        ELSIF (PositionsMoverPresent[1] > 0) AND
              (PositionsMoverPresent[2] = 0)
        THEN
          nCycleMover               :=   PositionsMoverPresent[1];
          nAxisFirst[nCycleMover]   :=   2;
          nCycle                    := 120;
        END_IF

      120:  // X=360 Y=120 --> 2
        IF  (PositionsMoverPresent[3] = 0) AND
            (PositionsMoverPresent[2] > 0)
        THEN
          nCycleMover               :=   PositionsMoverPresent[2];
          nAxisFirst[nCycleMover]   :=   2;
          nCycle                    := 130;

        ELSIF (PositionsMoverPresent[1] = 0) AND
              (PositionsMoverPresent[3] > 0)
        THEN
          nCycleMover               :=   PositionsMoverPresent[3];
          nAxisFirst[nCycleMover]   :=   0;
          nCycle                    := 110;
        END_IF

      130:  // X=360, Y=600 --> 3
        IF  (PositionsMoverPresent[3] = 0) AND
            (PositionsMoverPresent[2] > 0)
        THEN
          nCycleMover               :=   PositionsMoverPresent[2];
          nAxisFirst[nCycleMover]   :=   2;
          nCycle                    := 110;

        ELSIF (PositionsMoverPresent[3] > 0) AND
              (PositionsMoverPresent[1] > 0)
        THEN
          nCycleMover               :=   PositionsMoverPresent[1];
          nAxisFirst[nCycleMover]   :=   2;
          nCycle                    := 120;
        END_IF
    END_CASE
END_CASE
//-------------------------------------------------------------------------------------------------
// reset movers
//-------------------------------------------------------------------------------------------------
CASE nCycle
OF
  900:
    _bCyclePause                          :=
    _bCycleStop                           :=
    _bCycleStart                          := FALSE;

    MoverCtrl[1].Cmd                      := E_MOVER_CTRL.MOVER_RESET;

    IF (MoverState[1].State = E_MOVER_STATE.MOVER_RESET + E_PROGRESS.PROGRESS_DONE)
    THEN
      nCycle                              := 910;
      MoverCtrl[1].Cmd          := E_MOVER_CTRL.MOVER_NULL;

    ELSIF (MoverState[1].State = E_MOVER_STATE.MOVER_RESET + E_PROGRESS.PROGRESS_ERROR)
    THEN
      MoverCtrl[1].Cmd          := E_MOVER_CTRL.MOVER_NULL;
    END_IF

  910:
    MoverCtrl[2].Cmd                      := E_MOVER_CTRL.MOVER_RESET;

    IF (MoverState[2].State = E_MOVER_STATE.MOVER_RESET + E_PROGRESS.PROGRESS_DONE)
    THEN
      nCycle                              := 920;
      MoverCtrl[2].Cmd          := E_MOVER_CTRL.MOVER_NULL;

    ELSIF (MoverState[2].State = E_MOVER_STATE.MOVER_RESET + E_PROGRESS.PROGRESS_ERROR)
    THEN
      MoverCtrl[2].Cmd          := E_MOVER_CTRL.MOVER_NULL;
    END_IF

  920:
    MoverCtrl[1].Cmd                      := E_MOVER_CTRL.MOVER_DISABLE;

    IF (MoverState[1].State = E_MOVER_STATE.MOVER_DISABLE + E_PROGRESS.PROGRESS_DONE)
    THEN
      nCycle                              := 930;
      MoverCtrl[1].Cmd          := E_MOVER_CTRL.MOVER_NULL;
    END_IF

  930:
    MoverCtrl[2].Cmd                      := E_MOVER_CTRL.MOVER_DISABLE;

    IF (MoverState[2].State = E_MOVER_STATE.MOVER_DISABLE + E_PROGRESS.PROGRESS_DONE)
    THEN
      IF (_wCycleReset = 0)
      THEN
        nCycle                            := 0;
      ELSE
        nCycle                            := 1000;
      END_IF
      MoverCtrl[2].Cmd          := E_MOVER_CTRL.MOVER_NULL;
    END_IF
END_CASE
//-------------------------------------------------------------------------------------------------
// recovery procedure
//-------------------------------------------------------------------------------------------------
CASE nCycle
OF
  1000:
    _wCycleReset                          := 0;
    // position check
    // mover must be in position at any station
    IF  (PositionsMoverPresent[1] > 0) AND
        (PositionsMoverPresent[2] > 0)
    THEN
      nCycleMover                         := PositionsMoverPresent[2];
      MoveData[nCycleMover]               := Positions[3];
      nAxisFirst[nCycleMover]             := 2;

      MoverCtrl[1].Cmd                    := E_MOVER_CTRL.MOVER_ENABLE;
      MoverCtrl[2].Cmd                    := E_MOVER_CTRL.MOVER_ENABLE;
  
      IF (MoverState[1].State = E_MOVER_STATE.MOVER_ENABLE + E_PROGRESS.PROGRESS_DONE) AND
         (MoverState[2].State = E_MOVER_STATE.MOVER_ENABLE + E_PROGRESS.PROGRESS_DONE)
      THEN
        nCycle                        := 1010;
      ELSE
        IF (MoverInfo[1].bMoverError) OR
           (MoverInfo[2].bMoverError)
        THEN
          nCycle                      := 900;
        END_IF
      END_IF

    ELSIF (PositionsMoverPresent[1] > 0) AND
          (PositionsMoverPresent[3] > 0)
    THEN
      nCycleMover                         := PositionsMoverPresent[1];
      MoveData[nCycleMover]               := Positions[2];
      nAxisFirst[nCycleMover]             := 2;

      MoverCtrl[1].Cmd                := E_MOVER_CTRL.MOVER_ENABLE;
      MoverCtrl[2].Cmd                := E_MOVER_CTRL.MOVER_ENABLE;
  
      IF (MoverState[1].State = E_MOVER_STATE.MOVER_ENABLE + E_PROGRESS.PROGRESS_DONE) AND
         (MoverState[2].State = E_MOVER_STATE.MOVER_ENABLE + E_PROGRESS.PROGRESS_DONE)
      THEN
        nCycle                        := 1010;
      ELSE
        IF (MoverInfo[1].bMoverError) OR
           (MoverInfo[2].bMoverError)
        THEN
          nCycle                      := 900;
        END_IF
      END_IF


    ELSIF (PositionsMoverPresent[2] > 0) AND
          (PositionsMoverPresent[3] > 0)
    THEN
      nCycleMover                         := PositionsMoverPresent[3];
      MoveData[nCycleMover]               := Positions[1];
      nAxisFirst[nCycleMover]             := 2;

      MoverCtrl[1].Cmd                := E_MOVER_CTRL.MOVER_ENABLE;
      MoverCtrl[2].Cmd                := E_MOVER_CTRL.MOVER_ENABLE;
  
      IF (MoverState[1].State = E_MOVER_STATE.MOVER_ENABLE + E_PROGRESS.PROGRESS_DONE) AND
         (MoverState[2].State = E_MOVER_STATE.MOVER_ENABLE + E_PROGRESS.PROGRESS_DONE)
      THEN
        nCycle                        := 1010;
      ELSE
        IF (MoverInfo[1].bMoverError) OR
           (MoverInfo[2].bMoverError)
        THEN
          nCycle                      := 900;
        END_IF
      END_IF
    END_IF

  1010:
      MoverCtrl[nCycleMover].Cmd    := E_MOVER_CTRL.MOVER_MOVE_TO_POS;
      IF (MoverState[nCycleMover].State = E_MOVER_STATE.MOVER_MOVE_TO_POS + E_PROGRESS.PROGRESS_ERROR)
      THEN
        nCycle                      := 900; // defaut error reaction: reset and switch off all movers

      ELSE
        IF (MoverState[nCycleMover].State = E_MOVER_STATE.MOVER_MOVE_TO_POS + E_PROGRESS.PROGRESS_DONE)
        THEN
          nCycle                    := 0;
        END_IF
      END_IF
END_CASE 
//-------------------------------------------------------------------------------------------------
//-------------------------------------------------------------------------------------------------
//-------------------------------------------------------------------------------------------------
//-------------------------------------------------------------------------------------------------
IF (_bClearAllAlarms)
THEN
  _bClearAllAlarms                  := FALSE;
  _hrEventLog                       := fbEventLogger.ClearAllAlarms(0, TRUE);
END_IF
//-------------------------------------------------------------------------------------------------
//-------------------------------------------------------------------------------------------------
IF (_bClearLoggedEvents)
THEN
  _bClearLoggedEvents               := fbEventLogger.ClearLoggedEvents(0);
END_IF
//-------------------------------------------------------------------------------------------------
//-------------------------------------------------------------------------------------------------
//-------------------------------------------------------------------------------------------------
//-------------------------------------------------------------------------------------------------

METHOD MoverInPositionXY : BOOL   // checks if XY position matches mover position
VAR_INPUT
  nMover              : DINT;
  stPosition          : ST_POS_XYC;
  rDelta              : ARRAY[1..2] OF LREAL;      // target window for X and Y
END_VAR
VAR
  bInPosition_X,
  bInPosition_Y       : BOOL;
END_VAR
VAR
//  rModPosC            : ARRAY[1..MAX_XPLANAR_MOVERS] OF LREAL;
END_VAR

IF NOT (nMover > 0) OR
   NOT (nMover < MAX_XPLANAR_MOVERS+1)
THEN
  RETURN;
END_IF


bInPosition_X         :=    (MoverInfo[nMover].rActPosX > stPosition.x - rDelta[1]) 
                        AND (MoverInfo[nMover].rActPosX < stPosition.x + rDelta[1]);

bInPosition_Y         :=    (MoverInfo[nMover].rActPosY > stPosition.y - rDelta[2]) 
                        AND (MoverInfo[nMover].rActPosY < stPosition.y + rDelta[2]);

rModPosC[nMover]      := Tc2_Math.LMOD(MoverInfo[nMover].rActPosC, 90.0);

IF (bInPosition_X AND bInPosition_Y)
THEN
  IF ((rModPosC[nMover]) <   5) AND
     ((rModPosC[nMover]) >  -5)
  THEN
    MoverInPositionXY := TRUE;
  ELSIF (ABS(rModPosC[nMover]) < 95) AND
        (ABS(rModPosC[nMover]) > 85)
  THEN
    MoverInPositionXY := TRUE;
  END_IF
END_IF
END_METHOD

END_PROGRAM

// ---- Mover/fb_MoverCtrl.TcPOU
//---------------------------------------------------------------------------------------------------------------
//
//  HAUD 2023.12.18
//
//  - XTS_TRAINING
//  - example project for setting up transport layer
//
//
//  fb_MoverCtrl
//  - accepts orders (E_MOVER_CTRL) via cyclic struct interface to execute
//  - interface struct  to extern control
//
//
//---------------------------------------------------------------------------------------------------------------
// This SOFTWARE is provided as an Exemple by THE PROVIDER "as is" and "with all faults." THE PROVIDER makes no 
// representations or warranties of any kind concerning the safety, suitability, lack of viruses, inaccuracies, 
// typographical errors, or other harmful components of this SOFTWARE. There are inherent dangers in the use of 
// any software, and you are solely responsible for determining whether this SOFTWARE is compatible with your 
// equipment and other software installed on your equipment. You are also solely responsible for the protection 
// of your equipment and backup of your data, and THE PROVIDER will not be liable for any damages you may suffer 
// in connection with using, modifying, or distributing this SOFTWARE.
//---------------------------------------------------------------------------------------------------------------
FUNCTION_BLOCK fb_MoverCtrl EXTENDS fb_Mover
VAR
  // Ctrl and State for executing commands
  _stCtrl           : REFERENCE TO ARRAY[1..MAX_XPLANAR_MOVERS] OF ST_MOVER_CTRL;
  _stState          : REFERENCE TO ARRAY[1..MAX_XPLANAR_MOVERS] OF ST_MOVER_STATE;

  // data structures to use with commands
  _stMoveData       : REFERENCE TO ARRAY[1..MAX_XPLANAR_MOVERS] OF ST_MOVE_DATA;

  // external setpoint generator access to mover
	_pAxis            : POINTER TO ARRAY[1..3] OF AXIS_REF;

  // we are handling virtual axis, that need to be switched on
  _fbPower          : ARRAY[1..3] OF Tc2_MC2.MC_Power;
  _fbReset          : ARRAY[1..3] OF Tc2_MC2.MC_Reset;
  _fbSetPos         : ARRAY[1..3] OF Tc2_MC2.MC_SetPosition; // position is set to 0.0 because the setpoint generator here is hardcoded to relative movement

  // AXIS_REFs are feeding into here
	_stPosVector,
	_stVeloVector,
	_stAccVector		  : MoverVector;	

  _Extfeedback      : MC_PlanarFeedback;
  _ExtOptions       : ST_ExternalSetpointGenerationOptions;

  _eCmd,
  _eCmdOld          : E_MOVER_CTRL;

  _eState           : E_MOVER_STATE;

  _eResult          : E_PROGRESS;
END_VAR

IF NOT Check() THEN RETURN; END_IF

// copy to local for debug
_eCmd                         := _stCtrl[_nMoverId].Cmd;

// cyclic check for command change
// get state for cmd
IF (_eCmd <> _eCmdOld)
THEN
  // get matching sdtate for Ctrl.Cmd
  _eState                     := Cmd(_eCmd);
  _eCmdOld                    := _eCmd;
END_IF


CASE _eResult
OF
  E_PROGRESS.PROGRESS_INVALID:
    _stState[_nMoverId].State := E_MOVER_STATE.MOVER_NULL;

  E_PROGRESS.PROGRESS_ERROR:
    _stState[_nMoverId].State := _eState + E_PROGRESS.PROGRESS_ERROR;

  E_PROGRESS.PROGRESS_DONE:
    _stState[_nMoverId].State := _eState + E_PROGRESS.PROGRESS_DONE;

ELSE
  // work in progress
  // update progress for extern use
  _stState[_nMoverId].State   := _eState + _eResult;

  CASE _eState
  OF
    E_MOVER_STATE.MOVER_ENABLE:
      _eResult                := Enable(TRUE);
  
    E_MOVER_STATE.MOVER_DISABLE:
      _eResult                := Disable(TRUE);
  
    E_MOVER_STATE.MOVER_MOVE_TO_POS:
      _eResult                := MoveToPos(TRUE, _stMoveData[_nMoverId]);
  
    E_MOVER_STATE.MOVER_HALT:
      _eResult                := Halt(TRUE, _stMoveData[_nMoverId]);
  
    E_MOVER_STATE.MOVER_RESET:
      _eResult                := Reset(TRUE);

    E_MOVER_STATE.MOVER_EXT_DISABLE_AXIS:
      _eResult          := Ext_DisableAxis(TRUE);
  
    E_MOVER_STATE.MOVER_EXT_ENABLE_AXIS:
      _eResult          := Ext_EnableAxis(TRUE);
  
    E_MOVER_STATE.MOVER_EXT_SET_POSITION:
      _eResult          := Ext_SetPosition(TRUE);
  
    E_MOVER_STATE.MOVER_EXT_START:
      _eResult          := Ext_StartExtSetpointRelative(TRUE);
  
    E_MOVER_STATE.MOVER_EXT_STOP:
      _eResult          := Ext_StopExtSetpoint(TRUE);

  ELSE
      _eResult                := E_PROGRESS.PROGRESS_INVALID;
  END_CASE
END_CASE

METHOD PRIVATE Check : BOOL
// The thing that should not be

IF NOT (_nMoverId > 0)
THEN
  _eCheck                     := E_MOVER_CHECK.MOVER_ID_INVALID;
  RETURN;
END_IF

IF NOT __ISVALIDREF(_Mover)
THEN
  _eCheck                     := E_MOVER_CHECK.REFERENCE_AXIS_REF_INVALID;
  RETURN;
END_IF

IF NOT __ISVALIDREF(_stInfo)
THEN
  _eCheck                     := E_MOVER_CHECK.REFERENCE_INFO_INVALID;
  RETURN;
END_IF

IF NOT __ISVALIDREF(_stMoveData)
THEN
  _eCheck                     := E_MOVER_CHECK.REFERENCE_MOVE_DATA_INVALID;
  RETURN;
END_IF

IF NOT __ISVALIDREF(_stCtrl)
THEN
  _eCheck                     := E_MOVER_CHECK.REFERENCE_CTRL_INVALID;
  RETURN;
END_IF

IF NOT __ISVALIDREF(_stState)
THEN
  _eCheck                     := E_MOVER_CHECK.REFERENCE_STATE_INVALID;
  RETURN;
END_IF

IF NOT (_pAxis <> 0)
THEN
  _eCheck                     := E_MOVER_CHECK.POINTER_NCI_AXIS_REF_INVALID;
  RETURN;
END_IF


_eCheck                       := E_MOVER_CHECK.CHECK_DONE;
Check                         := TRUE;
END_METHOD

METHOD PRIVATE Cmd : E_MOVER_STATE
VAR_INPUT
  Ctrl      : E_MOVER_CTRL;
END_VAR
VAR_INST
  _eState   : E_MOVER_STATE;
END_VAR
IF NOT Check() THEN Cmd := E_MOVER_STATE.MOVER_NULL;  RETURN; END_IF


CASE Ctrl
OF
  E_MOVER_CTRL.MOVER_ENABLE:
    _eResult          := Enable(FALSE);
    _eState           := E_MOVER_STATE.MOVER_ENABLE;

  E_MOVER_CTRL.MOVER_DISABLE:
    _eResult          := Disable(FALSE);
    _eState           := E_MOVER_STATE.MOVER_DISABLE;

  E_MOVER_CTRL.MOVER_MOVE_TO_POS:
    _eResult          := MoveToPos(FALSE, _stMoveData[_nMoverId]);
    _eState           := E_MOVER_STATE.MOVER_MOVE_TO_POS;

  E_MOVER_CTRL.MOVER_HALT:
    _eResult          := Halt(FALSE, _stMoveData[_nMoverId]);
    _eState           := E_MOVER_STATE.MOVER_HALT;

  E_MOVER_CTRL.MOVER_RESET:
    _eResult          := Reset(FALSE);
    _eState           := E_MOVER_STATE.MOVER_RESET;

  E_MOVER_CTRL.MOVER_EXT_DISABLE_AXIS:
    _eResult          := Ext_DisableAxis(FALSE);
    _eState           := E_MOVER_STATE.MOVER_EXT_DISABLE_AXIS;

  E_MOVER_CTRL.MOVER_EXT_ENABLE_AXIS:
    _eResult          := Ext_EnableAxis(FALSE);
    _eState           := E_MOVER_STATE.MOVER_EXT_ENABLE_AXIS;

  E_MOVER_CTRL.MOVER_EXT_SET_POSITION:
    _eResult          := Ext_SetPosition(FALSE);
    _eState           := E_MOVER_STATE.MOVER_EXT_SET_POSITION;

  E_MOVER_CTRL.MOVER_EXT_START:
    _eResult          := Ext_StartExtSetpointRelative(FALSE);
    _eState           := E_MOVER_STATE.MOVER_EXT_START;

  E_MOVER_CTRL.MOVER_EXT_STOP:
    _eResult          := Ext_StopExtSetpoint(FALSE);
    _eState           := E_MOVER_STATE.MOVER_EXT_STOP;


ELSE
    _eResult          := E_PROGRESS.PROGRESS_INVALID; 
    _eState           := E_MOVER_STATE.MOVER_NULL;
END_CASE

Cmd                   := _eState;
END_METHOD

PROPERTY Ctrl : REFERENCE TO ARRAY[1..MAX_XPLANAR_MOVERS] OF ST_MOVER_CTRL
SET
_stCtrl ref= Ctrl;
END_SET
END_PROPERTY

METHOD Ext_DisableAxis : e_progress // disable the NCI AXIS_REF _pAxis[]
VAR_INPUT
  execute   : BOOL;
END_VAR
VAR_INST
  _nAxis    : uint;
  _nErrorId : UDINT;
  _idx      : UINT;
  _eState   : e_progress;
END_VAR
IF NOT Execute THEN _eState  := E_PROGRESS.PROGRESS_INIT; END_IF 
IF NOT Check() THEN Ext_DisableAxis  := E_PROGRESS.PROGRESS_ERROR; RETURN; END_IF


CASE _eState
OF
  E_PROGRESS.PROGRESS_INIT:
    IF Execute
    THEN
      _nErrorId               := 0;
      _nAxis                  := 1;
      _eState                 := E_PROGRESS.PROGRESS_BUSY;
    END_IF
END_CASE
//-----------------------------------------------------------------------------
//-----------------------------------------------------------------------------
CASE _eState
OF
  E_PROGRESS.PROGRESS_BUSY:
    _fbPower[_nAxis].Enable   := FALSE;

    IF NOT (_pAxis^[_nAxis].Status.ControlLoopClosed)
    THEN
      _eState                 := E_PROGRESS.PROGRESS_PREPARE;
    END_IF
    FOR _idx := 1 TO 3
    DO
      _pAxis^[_idx]();
      _fbPower[_idx](
              Axis:= _pAxis^[_idx], 
              Enable:= FALSE, 
              Enable_Positive:= TRUE, 
              Enable_Negative:= TRUE, 
              Override:= , 
              BufferMode:= , 
              Options:= , 
              Status=> , 
              Busy=> , 
              Error=> , 
              ErrorID=> _nErrorId);
    END_FOR

 END_CASE
//-----------------------------------------------------------------------------
//-----------------------------------------------------------------------------
CASE _eState
OF
  E_PROGRESS.PROGRESS_PREPARE:
    IF (_nAxis > 2)
    THEN
      _eState                 := E_PROGRESS.PROGRESS_DONE;
    ELSE
      _nAxis                  := _nAxis + 1;
      _eState                 := E_PROGRESS.PROGRESS_BUSY;
    END_IF
END_CASE
//-----------------------------------------------------------------------------
//-----------------------------------------------------------------------------

Ext_DisableAxis                       := _eState;
END_METHOD

METHOD Ext_EnableAxis : e_progress // enable the NCI AXIS_REF _pAxis[]
VAR_INPUT
  execute   : BOOL;
END_VAR
VAR_INST
  _nAxis    : uint;
  _nErrorId : UDINT;
  _idx      : UINT;
  _eState   : e_progress;
END_VAR
IF NOT Execute THEN _eState  := E_PROGRESS.PROGRESS_INIT; END_IF 
IF NOT Check() THEN Ext_EnableAxis  := E_PROGRESS.PROGRESS_ERROR; RETURN; END_IF


CASE _eState
OF
  E_PROGRESS.PROGRESS_INIT:
    IF Execute
    THEN
      _nErrorId               := 0;
      _nAxis                  := 1;
      _eState                 := E_PROGRESS.PROGRESS_BUSY;
    END_IF
END_CASE
//-----------------------------------------------------------------------------
//-----------------------------------------------------------------------------
CASE _eState
OF
  E_PROGRESS.PROGRESS_BUSY:
    _fbPower[_nAxis].Enable   := TRUE;

    IF (_pAxis^[_nAxis].Status.ControlLoopClosed)
    THEN
      _eState                 := E_PROGRESS.PROGRESS_PREPARE;
    END_IF
    FOR _idx := 1 TO 3
    DO
      _pAxis^[_idx]();
      _fbPower[_idx](
              Axis:= _pAxis^[_idx], 
              Enable:= TRUE, 
              Enable_Positive:= TRUE, 
              Enable_Negative:= TRUE, 
              Override:= 100.0, 
              BufferMode:= , 
              Options:= , 
              Status=> , 
              Busy=> , 
              Error=> , 
              ErrorID=> _nErrorId);
    END_FOR

 END_CASE
//-----------------------------------------------------------------------------
//-----------------------------------------------------------------------------
CASE _eState
OF
  E_PROGRESS.PROGRESS_PREPARE:
    IF (_nAxis > 2)
    THEN
      _eState                 := E_PROGRESS.PROGRESS_DONE;
    ELSE
      _nAxis                  := _nAxis + 1;
      _eState                 := E_PROGRESS.PROGRESS_BUSY;
    END_IF
END_CASE
//-----------------------------------------------------------------------------
//-----------------------------------------------------------------------------

Ext_EnableAxis                       := _eState;
END_METHOD

METHOD Ext_SetPosition : e_progress
VAR_INPUT
  Execute             : BOOL;
END_VAR
VAR_INST
  _rSetPos            : ARRAY[1..3] OF LREAL;
  _ndx                : udint;
  _nAxis              : UDINT;
  _nErrorId           : UDINT;
  _eState             : E_PROGRESS;
END_VAR
IF NOT Execute THEN _eState  := E_PROGRESS.PROGRESS_INIT; END_IF 
IF NOT Check() THEN Ext_SetPosition   := E_PROGRESS.PROGRESS_ERROR; RETURN; END_IF


CASE _eState
OF
  E_PROGRESS.PROGRESS_INIT:
    IF Execute
    THEN
      _rSetPos[1]               := 0.0; // these are hardcoded because the setpoint generator is set to relative movement
      _rSetPos[2]               := 0.0;
      _rSetPos[3]               := 0.0;

      _nErrorId                 := 0;
      _nAxis                    := 1;
      _eState                   := E_PROGRESS.PROGRESS_BUSY;

      FOR _ndx := 1 TO 3
      DO
        _fbSetPos[_ndx](
                    Axis:= _pAxis^[_ndx], 
                    Execute:= FALSE, 
                    Position:= 0.0);
      END_FOR
    END_IF
END_CASE
//-----------------------------------------------------------------------------
//-----------------------------------------------------------------------------
CASE _eState
OF
  E_PROGRESS.PROGRESS_BUSY:
    _fbSetPos[_nAxis](
                Axis:= _pAxis^[_nAxis], 
                Execute:= TRUE, 
                Position:= _rSetPos[_nAxis], 
                Mode:= , 
                Options:= , 
                Done=> , 
                Busy=> , 
                Error=> , 
                ErrorID=> );

    IF _fbSetPos[_nAxis].Done
    THEN
      _eState                 := E_PROGRESS.PROGRESS_PREPARE;
      _fbSetPos[_nAxis](
                Axis:= _pAxis^[_nAxis], 
                Execute:= FALSE);
    END_IF 

  E_PROGRESS.PROGRESS_PREPARE:
    IF (_nAxis > 2)
    THEN
      _eState                 := E_PROGRESS.PROGRESS_DONE;
    ELSE
      _nAxis                  := _nAxis + 1;
      _eState                 := E_PROGRESS.PROGRESS_BUSY;
    END_IF
END_CASE
//-----------------------------------------------------------------------------
//-----------------------------------------------------------------------------
CASE _eState
OF
  E_PROGRESS.PROGRESS_STARTUP:

  E_PROGRESS.PROGRESS_CHECK:
    _eState                     := E_PROGRESS.PROGRESS_OCCUPIED;

END_CASE
//-----------------------------------------------------------------------------
//-----------------------------------------------------------------------------
CASE _eState
OF
  E_PROGRESS.PROGRESS_OCCUPIED:

END_CASE
//-----------------------------------------------------------------------------
//-----------------------------------------------------------------------------
CASE _eState
OF
  E_PROGRESS.PROGRESS_WORKING:
END_CASE
//-----------------------------------------------------------------------------
//-----------------------------------------------------------------------------
CASE _eState
OF
  E_PROGRESS.PROGRESS_STILL_WORKING:
END_CASE
//-----------------------------------------------------------------------------
//-----------------------------------------------------------------------------
Ext_SetPosition                       := _eState;
//-----------------------------------------------------------------------------
//-----------------------------------------------------------------------------
END_METHOD

METHOD Ext_StartExtSetpointRelative : e_progress
VAR_INPUT
  Execute   : BOOL;
END_VAR
VAR_INST
  _nAxis    : uint;
  _nErrorId : UDINT;
  _idx      : UINT;
  _eState   : e_progress;
END_VAR
IF NOT Execute THEN _eState                       := E_PROGRESS.PROGRESS_INIT; END_IF 
IF NOT Check() THEN Ext_StartExtSetpointRelative  := E_PROGRESS.PROGRESS_ERROR; RETURN; END_IF


CASE _eState
OF
  E_PROGRESS.PROGRESS_INIT:
    IF Execute
    THEN
      _nErrorId               := 0;
      _nAxis                  := 1;
      _eState                 := E_PROGRESS.PROGRESS_BUSY;
      _ExtOptions.mode        := MC_EXTERNAL_SET_POSITION_MODE.Relative;  // this example runs with relative movement
    END_IF
END_CASE
//-----------------------------------------------------------------------------
//-----------------------------------------------------------------------------
CASE _eState
OF
  E_PROGRESS.PROGRESS_BUSY:
    _Mover.StartExternalSetpointGeneration(_Extfeedback,_ExtOptions);
    _eState                   := E_PROGRESS.PROGRESS_PREPARE;
END_CASE
//-----------------------------------------------------------------------------
//-----------------------------------------------------------------------------
CASE _eState
OF
  E_PROGRESS.PROGRESS_PREPARE:
    _Extfeedback.Update();

    IF (_Extfeedback.Done)
    THEN
      _eState                 := E_PROGRESS.PROGRESS_WORKING;

    ELSIF (_Extfeedback.Aborted) OR
          (_Extfeedback.Error)
    THEN
      _nErrorId               := _Extfeedback.ErrorId;
      _eState                 := E_PROGRESS.PROGRESS_ERROR;
    END_IF
END_CASE
//-----------------------------------------------------------------------------
//-----------------------------------------------------------------------------
CASE _eState
OF
  E_PROGRESS.PROGRESS_working:
    FOR _idx := 1 TO 3
    DO
      _pAxis^[_idx]();
      _fbPower[_idx](
            Axis              := _pAxis^[_idx], 
            Enable_Positive   := TRUE, 
            Enable_Negative   := TRUE, 
            Override          := , 
            BufferMode        := , 
            Options           := , 
            Status            => , 
            Busy              => , 
            Error             => , 
            ErrorID           => );
    END_FOR

    _stPosVector.x 	          := _pAxis^[1].NcToPlc.SetPos;
    _stVeloVector.x	          := _pAxis^[1].NcToPlc.SetVelo;
    _stAccVector.x		        := _pAxis^[1].NcToPlc.SetAcc;
  
    _stPosVector.y 	          := _pAxis^[2].NcToPlc.SetPos;
    _stVeloVector.y	          := _pAxis^[2].NcToPlc.SetVelo;
    _stAccVector.y		        := _pAxis^[2].NcToPlc.SetAcc;
  
    _stPosVector.z 	          := _pAxis^[3].NcToPlc.SetPos;
    _stVeloVector.z	          := _pAxis^[3].NcToPlc.SetVelo;
    _stAccVector.z		        := _pAxis^[3].NcToPlc.SetAcc;
  
    _Mover.SetExternalSetpoint(_stPosVector, _stVeloVector, _stAccVector);
    _Mover.Update();
 END_CASE
//-----------------------------------------------------------------------------
//-----------------------------------------------------------------------------

Ext_StartExtSetpointRelative  := _eState;
END_METHOD

METHOD Ext_StopExtSetpoint : e_progress
VAR_INPUT
  Execute   : Bool;
END_VAR
VAR_INST
  _nAxis    : uint;
  _nErrorId : UDINT;
  _idx      : UINT;
  _eState   : e_progress;
END_VAR
IF NOT Execute THEN _eState               := E_PROGRESS.PROGRESS_INIT; END_IF 
IF NOT Check() THEN Ext_StopExtSetpoint   := E_PROGRESS.PROGRESS_ERROR; RETURN; END_IF


CASE _eState
OF
  E_PROGRESS.PROGRESS_INIT:
    IF Execute
    THEN
      _nErrorId               := 0;
      _nAxis                  := 1;
      _eState                 := E_PROGRESS.PROGRESS_BUSY;
    END_IF
END_CASE
//-----------------------------------------------------------------------------
//-----------------------------------------------------------------------------
CASE _eState
OF
  E_PROGRESS.PROGRESS_BUSY:
    _Mover.StopExternalSetpointGeneration(_Extfeedback);
    _eState                   := E_PROGRESS.PROGRESS_PREPARE;
END_CASE
//-----------------------------------------------------------------------------
//-----------------------------------------------------------------------------
CASE _eState
OF
  E_PROGRESS.PROGRESS_PREPARE:
    _Extfeedback.Update();

    IF (_Extfeedback.Done)
    THEN
      _eState               := E_PROGRESS.PROGRESS_DONE;

    ELSIF (_Extfeedback.Aborted) OR
          (_Extfeedback.Error)
    THEN
      _nErrorId             := _Extfeedback.ErrorId;
      _eState               := E_PROGRESS.PROGRESS_ERROR;
    END_IF
END_CASE
//-----------------------------------------------------------------------------
//-----------------------------------------------------------------------------

Ext_StopExtSetpoint         := _eState;
END_METHOD

PROPERTY MoveData : reference TO ARRAY[1..MAX_XPLANAR_MOVERS] OF st_move_data
SET
_stMoveData REF= MoveData;
END_SET
END_PROPERTY

PROPERTY pAxis : pointer to array[1..3] of AXIS_REF
SET
_pAxis := pAxis;
END_SET
END_PROPERTY

PROPERTY State : REFERENCE TO ARRAY[1..MAX_XPLANAR_MOVERS] OF ST_MOVER_STATE
SET
_stState ref= State;
END_SET
END_PROPERTY

END_FUNCTION_BLOCK

// ---- Mover/fb_Mover.TcPOU
//---------------------------------------------------------------------------------------------------------------
//
//  HAUD 2024.04.16
//
//
//
//---------------------------------------------------------------------------------------------------------------
// This SOFTWARE is provided as an Exemple by THE PROVIDER "as is" and "with all faults." THE PROVIDER makes no 
// representations or warranties of any kind concerning the safety, suitability, lack of viruses, inaccuracies, 
// typographical errors, or other harmful components of this SOFTWARE. There are inherent dangers in the use of 
// any software, and you are solely responsible for determining whether this SOFTWARE is compatible with your 
// equipment and other software installed on your equipment. You are also solely responsible for the protection 
// of your equipment and backup of your data, and THE PROVIDER will not be liable for any damages you may suffer 
// in connection with using, modifying, or distributing this SOFTWARE.
//---------------------------------------------------------------------------------------------------------------
FUNCTION_BLOCK fb_Mover
VAR
  _eCheck           : E_MOVER_CHECK;
  _nMoverId         : UINT;

  _Mover            : REFERENCE TO Tc3_Mc3PlanarMotion.MC_PlanarMover;
  _Feedback         : REFERENCE TO Tc3_Mc3PlanarMotion.MC_PlanarFeedback;

  // mover compact axis information
  _stInfo           : REFERENCE TO ST_MOVER_INFO; // ActPos, Enable, ...

  _bError           : BOOL;   // used in Cycle()
  _nErrorIdMover,             // used in Cycle()
  _nErrorIdPower    : UDINT;  // used in Cycle()

  //---------------------------------------------------------------------------
  // 
  //---------------------------------------------------------------------------
  _wMoverState      : DWORD;

END_VAR

METHOD Check : BOOL
// check The thing that should not be

IF NOT (_nMoverId > 0)
THEN
  _eCheck                     := E_MOVER_CHECK.MOVER_ID_INVALID;
  RETURN;
END_IF

IF NOT __ISVALIDREF(_Mover)
THEN
  _eCheck                     := E_MOVER_CHECK.REFERENCE_AXIS_REF_INVALID;
  RETURN;
END_IF

IF NOT __ISVALIDREF(_stInfo)
THEN
  _eCheck                     := E_MOVER_CHECK.REFERENCE_INFO_INVALID;
  RETURN;
END_IF

_eCheck                       := E_MOVER_CHECK.CHECK_DONE;
Check                         := TRUE;
END_METHOD

METHOD Cycle : E_PROGRESS
VAR_INST
  _eState             : E_PROGRESS;

  _rtrigMoverError,
  _rtrigPowerError    : Tc2_Standard.R_TRIG;
END_VAR
IF NOT Check() THEN Cycle := E_PROGRESS.PROGRESS_ERROR; RETURN; END_IF

//-----------------------------------------------------------------------------------------------
// cyclic NC mapping
//-----------------------------------------------------------------------------------------------
_Mover.Update();
_Feedback.Update();
//-----------------------------------------------------------------------------------------------


//-----------------------------------------------------------------------------------------------
// cyclic error
//-----------------------------------------------------------------------------------------------

_rtrigPowerError(CLK := _Feedback.Error);

IF _rtrigMoverError.Q
THEN
  _bError                 := TRUE;  // deleted by Reset()
  // catch error
  _nErrorIdMover          := _Feedback.ErrorId;
  _stInfo.nErrorId        := _nErrorIdMover;
END_IF
//-----------------------------------------------------------------------------------------------

//-----------------------------------------------------------------------------------------------
// cyclic state
//-----------------------------------------------------------------------------------------------
IF NOT (_Mover.MCTOPLC.STD.State = MC_PLANAR_STATE.Enabled)
THEN
  _eState                       := E_PROGRESS.PROGRESS_INIT;
ELSE
  _eState                       := E_PROGRESS.PROGRESS_WORKING;
END_IF
 
IF _bError
THEN
  _eState                       := E_PROGRESS.PROGRESS_ERROR;
END_IF
//-----------------------------------------------------------------------------------------------


//-----------------------------------------------------------------------------
// cyclic Mover info data
// get collision avoiding information from cyclic interface
//-----------------------------------------------------------------------------------------------
_stInfo.bMoverEnabled           := (_Mover.MCTOPLC.STD.State = MC_PLANAR_STATE.Enabled);
_stInfo.bMoverStandstill        := NOT (_Mover.MCTOPLC.STD.Busy.BusyXYC);
_stInfo.bMoverError             := _bError;

_stInfo.rActPos.x               := _Mover.MCTOPLC.ACT.ActPos.x;
_stInfo.rActPos.y               := _Mover.MCTOPLC.ACT.ActPos.y;
_stInfo.rActPos.c               := _Mover.MCTOPLC.ACT.ActPos.c;
                                
_stInfo.rActPosX                := _Mover.MCTOPLC.ACT.ActPos.x;
_stInfo.rActPosY                := _Mover.MCTOPLC.ACT.ActPos.y;
_stInfo.rActPosC                := _Mover.MCTOPLC.ACT.ActPos.c;
                                
_stInfo.rActPosZ                := _Mover.MCTOPLC.ACT.ActPos.z;
                                
_stInfo.rActVeloX               := _Mover.MCTOPLC.ACT.ActVelo.x;
_stInfo.rActVeloY               := _Mover.MCTOPLC.ACT.ActVelo.y;
_stInfo.rActVeloZ               := _Mover.MCTOPLC.ACT.ActVelo.z;
_stInfo.rActVeloC               := _Mover.MCTOPLC.ACT.ActVelo.c;
//-----------------------------------------------------------------------------

Cycle                           := _eState;
END_METHOD

METHOD Disable : E_PROGRESS
VAR_INPUT
  Execute             : BOOL;
END_VAR
VAR_INST
  _nErrorId           : UDINT;
  _eState             : E_PROGRESS;
END_VAR
IF NOT Execute THEN _eState  := E_PROGRESS.PROGRESS_INIT; END_IF 
IF NOT Check() THEN Disable  := E_PROGRESS.PROGRESS_ERROR; RETURN; END_IF


CASE _eState
OF
  E_PROGRESS.PROGRESS_INIT:
    IF Execute
    THEN
      _nErrorId               := 0;
      _eState                 := E_PROGRESS.PROGRESS_BUSY;
    END_IF
END_CASE
//-----------------------------------------------------------------------------
//-----------------------------------------------------------------------------
CASE _eState
OF
  E_PROGRESS.PROGRESS_BUSY:
    _eState                   := E_PROGRESS.PROGRESS_PREPARE;
    _Mover.Disable(_Feedback);
END_CASE
//-----------------------------------------------------------------------------
//-----------------------------------------------------------------------------
CASE _eState
OF
  E_PROGRESS.PROGRESS_PREPARE:
    IF (_Mover.MCTOPLC.STD.State = MC_PLANAR_STATE.Disabled)
    THEN
      IF _Feedback.Error
      THEN
        _eState                 := E_PROGRESS.PROGRESS_ERROR;
      ELSIF _Feedback.Done
      THEN
        _eState                 := E_PROGRESS.PROGRESS_DONE;
      END_IF
    END_IF
END_CASE
//-----------------------------------------------------------------------------
//-----------------------------------------------------------------------------

Disable                       := _eState;
END_METHOD

METHOD Enable : E_PROGRESS
VAR_INPUT
  Execute             : BOOL;
END_VAR
VAR_INST
  _nErrorId           : UDINT;
  _eState             : E_PROGRESS;
END_VAR
IF NOT Execute THEN _eState  := E_PROGRESS.PROGRESS_INIT; END_IF 
IF NOT Check() THEN Enable   := E_PROGRESS.PROGRESS_ERROR; RETURN; END_IF


CASE _eState
OF
  E_PROGRESS.PROGRESS_INIT:
    IF Execute
    THEN
      _nErrorId               := 0;
      _eState                 := E_PROGRESS.PROGRESS_BUSY;
    END_IF
END_CASE
//-----------------------------------------------------------------------------
//-----------------------------------------------------------------------------
CASE _eState
OF
  E_PROGRESS.PROGRESS_BUSY:
    _eState                   := E_PROGRESS.PROGRESS_PREPARE;
    _Mover.Enable(_Feedback);
END_CASE
//-----------------------------------------------------------------------------
//-----------------------------------------------------------------------------
CASE _eState
OF
  E_PROGRESS.PROGRESS_PREPARE:
    IF (_Mover.MCTOPLC.STD.State = MC_PLANAR_STATE.Enabled)
    THEN
      IF _Feedback.Error
      THEN
        _eState                 := E_PROGRESS.PROGRESS_ERROR;
      ELSIF _Feedback.Done
      THEN
        _eState                 := E_PROGRESS.PROGRESS_DONE;
      END_IF
    ELSIF (_Mover.MCTOPLC.STD.State = MC_PLANAR_STATE.Error)
    THEN
      _eState                   := E_PROGRESS.PROGRESS_ERROR;
    END_IF
END_CASE
//-----------------------------------------------------------------------------
//-----------------------------------------------------------------------------

Enable                   := _eState;
END_METHOD

PROPERTY Feedback : reference to Tc3_Mc3PlanarMotion.MC_PlanarFeedback
SET
_Feedback REF= Feedback;
END_SET
END_PROPERTY

METHOD Halt : E_PROGRESS
VAR_INPUT
  Execute             : BOOL;
  stMoveData          : ST_MOVE_DATA;
END_VAR
VAR_INST
  _nErrorId           : UDINT;
  _eState             : E_PROGRESS;

	_Position           : Tc3_Physics.PositionXYC;
	_Constraint         : Tc3_Physics.DynamicConstraint_PathXY;
	_Options            : Tc3_Mc3PlanarMotion.ST_MoveToPositionOptions;
	_OptionsC           : ST_MoveCOptions;
END_VAR
IF NOT Execute 
THEN 
	_eState := E_PROGRESS.PROGRESS_INIT; 
END_IF 
IF NOT Check() 
THEN 
	Halt := E_PROGRESS.PROGRESS_ERROR; 
	RETURN; 
END_IF


CASE _eState
OF
  E_PROGRESS.PROGRESS_INIT:
    IF Execute
    THEN
      _nErrorId               := 0;
      _eState                 := E_PROGRESS.PROGRESS_BUSY;
    END_IF
END_CASE
//-----------------------------------------------------------------------------
//-----------------------------------------------------------------------------
CASE _eState
OF
  E_PROGRESS.PROGRESS_BUSY:
    _eState                     := E_PROGRESS.PROGRESS_PREPARE;
		_Position.SetValuesXYC(
                            x   := stMoveData.rPos.x,
													  y   := stMoveData.rPos.y,
                            c	  := 0.0);
								
		_Constraint.SetValuesVADJ(
                            V   := stMoveData.rVelo, 
                            A   := stMoveData.rAcc, 
                            D   := stMoveData.rAcc, 
                            J   := stMoveData.rJerk);

		_Options.useOrientation	    := FALSE;
END_CASE
//-----------------------------------------------------------------------------
//-----------------------------------------------------------------------------
CASE _eState
OF
  E_PROGRESS.PROGRESS_PREPARE:
    _eState                     := E_PROGRESS.PROGRESS_STARTUP;
    _Mover.Halt(_Feedback, _Constraint); 
END_CASE
//-----------------------------------------------------------------------------
//-----------------------------------------------------------------------------
CASE _eState
OF
  E_PROGRESS.PROGRESS_STARTUP:
    IF _Feedback.Error
    THEN
      _nErrorId                 := _feedback.ErrorId;
      _stInfo.nErrorId          := _nErrorId;

      _eState                   := E_PROGRESS.PROGRESS_ERROR;
    ELSIF _Feedback.Done
    THEN
      _eState                   := E_PROGRESS.PROGRESS_DONE;
    END_IF
END_CASE
//-----------------------------------------------------------------------------
//-----------------------------------------------------------------------------

Halt                          := _eState;
END_METHOD

PROPERTY Mover : REFERENCE to Tc3_Mc3PlanarMotion.MC_PlanarMover
SET
_Mover REF= Mover;
END_SET
END_PROPERTY

PROPERTY MoverId : uint
SET
_nMoverId := MoverId;
END_SET
END_PROPERTY

PROPERTY MoverInfo : REFERENCE to ST_MOVER_INFO
SET


	_stInfo ref= MoverInfo;
END_SET
END_PROPERTY

METHOD MoveToPos : E_PROGRESS
VAR_INPUT
  Execute             : BOOL;
  stMoveData          : ST_MOVE_DATA;
END_VAR
VAR_INST
  _nErrorId           : UDINT;
  _rDelta,
  _rPos               : LREAL;
  _eState             : E_PROGRESS;

	_Position           : Tc3_Physics.PositionXYC;
	_Constraint         : Tc3_Physics.DynamicConstraint_PathXY;
  _ConstraintC        : Tc3_Physics.DynamicConstraint_PathXY;
	_Options            : Tc3_Mc3PlanarMotion.ST_MoveToPositionOptions;
	_OptionsC           : ST_MoveCOptions;

  _rTmpV,
  _rTmpA,
  _rTmpD,
  _rTmpJ              : LREAL;
END_VAR
IF NOT Execute THEN _eState  := E_PROGRESS.PROGRESS_INIT; END_IF 
IF NOT Check() THEN MoveToPos   := E_PROGRESS.PROGRESS_ERROR; RETURN; END_IF


CASE _eState
OF
  E_PROGRESS.PROGRESS_INIT:
    IF Execute
    THEN
      _nErrorId                 := 0;
      _rDelta                   := SEL((stMoveData.rDelta < 0.01), stMoveData.rDelta, 0.05);
      _eState                   := E_PROGRESS.PROGRESS_BUSY;

      _rTmpV   := stMoveData.rVelo/10.0; 
      _rTmpA   := stMoveData.rAcc/10.0;
      _rTmpD   := stMoveData.rAcc/10.0; 
      _rTmpJ   := stMoveData.rJerk/10.0;


		  _Constraint.SetValuesVADJ(
                            V   := _rTmpV, 
                            A   := _rTmpA, 
                            D   := _rTmpD, 
                            J   := _rTmpJ);
  
      _Mover.MoveZ(
            commandFeedback     := _Feedback, 
            targetPosition      := stMoveData.rPosZ,
            constraint          := _Constraint);

		  _Options.useOrientation	  := FALSE;
    END_IF
END_CASE
//-----------------------------------------------------------------------------
//-----------------------------------------------------------------------------
CASE _eState
OF
  E_PROGRESS.PROGRESS_BUSY:
    IF _Feedback.Error OR _Feedback.Aborted
    THEN
      _nErrorId                 := _feedback.ErrorId;
      _stInfo.nErrorId          := _nErrorId;

      _eState                   := E_PROGRESS.PROGRESS_ERROR;

    ELSIF _Feedback.Done OR NOT _Feedback.Busy
    THEN
      _eState                   := E_PROGRESS.PROGRESS_PREPARE;

      IF (stMoveData.nAxisFirst = 1)
      THEN
        _Position.SetValuesXYC(
                            x   := stMoveData.rPos.x,
                            y   := _Mover.MCTOPLC.SET.SetPos.y,
                            c	  := 0.0);

      ELSIF (stMoveData.nAxisFirst = 2)
      THEN
        _Position.SetValuesXYC(
                            x   := _Mover.MCTOPLC.SET.SetPos.x,
                            y   := stMoveData.rPos.y,
                            c	  := 0.0);
      ELSE
        _Position.SetValuesXYC(
                            x   := stMoveData.rPos.x,
                            y   := stMoveData.rPos.y,
                            c	  := 0.0);
      END_IF								

		  _Options.useOrientation	  := FALSE;
    END_IF

  E_PROGRESS.PROGRESS_PREPARE:
    _eState                     := E_PROGRESS.PROGRESS_STARTUP;
		  _Options.useOrientation	  := FALSE;

		  _Constraint.SetValuesVADJ(
                            V   := stMoveData.rVelo, 
                            A   := stMoveData.rAcc, 
                            D   := stMoveData.rAcc, 
                            J   := stMoveData.rJerk);


		_Mover.MoveToPosition(
            commandFeedback     := _Feedback, 
            targetPosition      := _Position, 
            constraint          := _Constraint, 
            options             := _Options);

END_CASE
//-----------------------------------------------------------------------------
//-----------------------------------------------------------------------------
CASE _eState
OF
  E_PROGRESS.PROGRESS_STARTUP:
    IF _Feedback.Error OR _Feedback.Aborted
    THEN
      _nErrorId                 := _Feedback.ErrorId;
      _stInfo.nErrorId          := _nErrorId;

      _eState                   := E_PROGRESS.PROGRESS_ERROR;

    ELSIF _Feedback.Done  OR NOT _Feedback.Busy
    THEN

      IF (stMoveData.nAxisFirst = 1)
      THEN
        _eState                 := E_PROGRESS.PROGRESS_CHECK;
        _Position.SetValuesXYC(
                            x   := _Mover.MCTOPLC.ACT.ActPos.x,
                            y   := stMoveData.rPos.y,
                            c	  := 0.0);

      ELSIF (stMoveData.nAxisFirst = 2)
      THEN
        _eState                 := E_PROGRESS.PROGRESS_CHECK;
        _Position.SetValuesXYC(
                            x   := stMoveData.rPos.x,
                            y   := _Mover.MCTOPLC.ACT.ActPos.y,
                            c	  := 0.0);
      ELSE
        _eState                 := E_PROGRESS.PROGRESS_WORKING;

      END_IF								

		  _Options.useOrientation	  := FALSE;
    END_IF

  E_PROGRESS.PROGRESS_CHECK:
    _eState                     := E_PROGRESS.PROGRESS_OCCUPIED;
		  _Options.useOrientation	  := FALSE;

		  _Constraint.SetValuesVADJ(
                            V   := stMoveData.rVelo, 
                            A   := stMoveData.rAcc, 
                            D   := stMoveData.rAcc, 
                            J   := stMoveData.rJerk);


		_Mover.MoveToPosition(
            commandFeedback     := _Feedback, 
            targetPosition      := _Position, 
            constraint          := _Constraint, 
            options             := _Options);

END_CASE
//-----------------------------------------------------------------------------
//-----------------------------------------------------------------------------
CASE _eState
OF
  E_PROGRESS.PROGRESS_OCCUPIED:
    IF _Feedback.Error OR _Feedback.Aborted
    THEN
      _nErrorId                 := _Feedback.ErrorId;
      _stInfo.nErrorId          := _nErrorId;

      _eState                   := E_PROGRESS.PROGRESS_ERROR;

    ELSIF _Feedback.Done OR NOT _Feedback.Busy
    THEN
      _eState                   := E_PROGRESS.PROGRESS_WORKING;
		  _Options.useOrientation	  := FALSE;
    END_IF
END_CASE
//-----------------------------------------------------------------------------
//-----------------------------------------------------------------------------
CASE _eState
OF
  E_PROGRESS.PROGRESS_WORKING:
    _eState                     := E_PROGRESS.PROGRESS_STILL_WORKING;

        _rTmpV   := stMoveData.rVelo/10.0; 
        _rTmpA   := stMoveData.rAcc/10.0;
        _rTmpD   := stMoveData.rAcc/10.0; 
        _rTmpJ   := stMoveData.rJerk/10.0;
  
        _ConstraintC.SetValuesVADJ(
                            V   := _rTmpV, 
                            A   := _rTmpA, 
                            D   := _rTmpD, 
                            J   := _rTmpJ);

    _OptionsC.additionalTurns   := 0;
    _OptionsC.direction         := stMoveData.rPos.cDirection;;

    _Mover.MoveC(
            commandFeedback     := _Feedback, 
            targetPosition      := stMoveData.rPos.c,
            constraint          := _ConstraintC,
            options             := _OptionsC);
END_CASE
//-----------------------------------------------------------------------------
//-----------------------------------------------------------------------------
CASE _eState
OF
  E_PROGRESS.PROGRESS_STILL_WORKING:
    IF _Feedback.Error OR _Feedback.Aborted
    THEN
      _nErrorId                 := _Feedback.ErrorId;
      _stInfo.nErrorId          := _nErrorId;

      _eState                   := E_PROGRESS.PROGRESS_ERROR;

    ELSIF _Feedback.Done OR NOT _Feedback.Busy
    THEN
      IF (_stInfo.rActPosC < stMoveData.rPos.c + 0.02) AND
         (_stInfo.rActPosC > stMoveData.rPos.c - 0.02)
      THEN
        _eState                  := E_PROGRESS.PROGRESS_DONE;
      END_IF
    END_IF
END_CASE
//-----------------------------------------------------------------------------
//-----------------------------------------------------------------------------
MoveToPos                       := _eState;
//-----------------------------------------------------------------------------
//-----------------------------------------------------------------------------
END_METHOD

METHOD Reset : E_PROGRESS
VAR_INPUT
  Execute             : BOOL;
END_VAR
VAR_INST
  _nErrorId           : UDINT;
  _eState             : E_PROGRESS;
END_VAR
IF NOT Execute THEN _eState  := E_PROGRESS.PROGRESS_INIT; END_IF 
IF NOT Check() THEN Reset    := E_PROGRESS.PROGRESS_ERROR; RETURN; END_IF


CASE _eState
OF
  E_PROGRESS.PROGRESS_INIT:
    IF Execute
    THEN
      _stInfo.nErrorId        :=
      _nErrorId               := 0;
      _eState                 := E_PROGRESS.PROGRESS_BUSY;
    END_IF
END_CASE
//-----------------------------------------------------------------------------
//-----------------------------------------------------------------------------
CASE _eState
OF
  E_PROGRESS.PROGRESS_BUSY:
    _eState                   := E_PROGRESS.PROGRESS_PREPARE;
    _Mover.Reset(_Feedback);
END_CASE
//-----------------------------------------------------------------------------
//-----------------------------------------------------------------------------
CASE _eState
OF
  E_PROGRESS.PROGRESS_PREPARE:
    IF _Feedback.Error
    THEN
      _nErrorId               := _Feedback.ErrorId;
      _stInfo.nErrorId        := _nErrorId;

      _eState                 := E_PROGRESS.PROGRESS_ERROR;

    ELSIF _Feedback.Done
    THEN
      _eState                 := E_PROGRESS.PROGRESS_DONE;
    END_IF
END_CASE
//-----------------------------------------------------------------------------
//-----------------------------------------------------------------------------

Reset                         := _eState;
END_METHOD

END_FUNCTION_BLOCK

// ---- misc/fb_Blink.TcPOU
FUNCTION_BLOCK fb_Blink
VAR_INPUT
	tLowTime		: TIME;
	tCycleTime	: TIME;
END_VAR
VAR_OUTPUT
	bCycle			: BOOL;
END_VAR
VAR
	tonLowTime		: TON;
	tofCycleTime	: TOF;
END_VAR

tonLowTime(IN:=(NOT tofCycleTime.Q), PT:= tLowTime);
tofCycleTime(IN:=(tonLowTime.Q), PT:= tCycleTime);

bCycle := tofCycleTime.Q;

END_FUNCTION_BLOCK

// ---- misc/fb_LocalTime.TcPOU
FUNCTION_BLOCK fb_LocalTime
VAR_INPUT

END_VAR
VAR_OUTPUT
  sLocalTime  : STRING;
  dtLocalTime : DT;
END_VAR
VAR
  GetSysTime    : FW_GetSystemTime;
  strFileTime   : Tc2_Utilities.T_FILETIME;
END_VAR

GetSysTime(dwTimeLo=> strFileTime.dwLowDateTime, dwTimeHi=> strFileTime.dwHighDateTime);

sLocalTime := SYSTEMTIME_TO_STRING( FILETIME_TO_SYSTEMTIME( strFileTime ) );
dtLocalTime := systemtime_to_dt( FILETIME_TO_SYSTEMTIME( strFileTime ) );

END_FUNCTION_BLOCK

// ---- misc/f_DelBit64.TcPOU
FUNCTION f_DelBit64 : LWORD
VAR_INPUT
	inVal		: LWORD;
	bitNo		: DINT;
END_VAR
VAR
	wConst : LWORD := 1;
END_VAR

IF ( inVal AND SHL( wConst,bitNo MOD 64 ) ) > 0 THEN
	f_DelBit64 := inVal XOR (SHL( wConst,bitNo MOD 64 ));
ELSE
	f_DelBit64 := inVal;
END_IF

END_FUNCTION

// ---- misc/f_GetBit64.TcPOU
FUNCTION f_GetBit64 : bool
VAR_INPUT
  lwIn      : LWORD;
  bitNo     : INT;
END_VAR
VAR
  lwConst   : LWORD := 1;
END_VAR

IF ( lwIn AND SHL( lwConst,INT_TO_SINT(bitNo) MOD 64 ) ) > 0
THEN
  f_GetBit64 := TRUE;
ELSE
  f_GetBit64 := FALSE;
END_IF

END_FUNCTION

// ---- misc/f_GetBools.TcPOU
FUNCTION f_GetBools : LWORD
VAR_INPUT
  pArr    : POINTER TO BYTE;
  nLow    : DINT;
  nUp     : DINT;
END_VAR
VAR
  _idx    : DINT;
  _pData  : POINTER TO BYTE;
  _wRet   : LWORD;
END_VAR

FOR _idx := 0 TO nUp-1
DO
  _pData := pArr;
  IF NOT(_idx < nLow-1)
  THEN
    IF (_pData^ = 1)
    THEN
      _wRet := f_Setbit64(_wRet, _idx);
    END_IF
  END_IF
  pArr := pArr + 1;
END_FOR
f_GetBools := _wRet;

END_FUNCTION

// ---- misc/f_Setbit64.TcPOU
FUNCTION f_Setbit64 : LWORD
VAR_INPUT
	inVal		: LWORD;
	bitNo		: DINT;
END_VAR
VAR
	wConst	: LWORD := 1;
END_VAR

f_Setbit64 := inVal OR SHL( wConst,bitNo MOD 64 );

END_FUNCTION

// ---- GlobalTextList.TcGTLO
TEXTLIST GlobalTextList
  300 = '%i'
  77 = 'Aborting'
  44 = 'Again'
  24 = 'CycleStop'
  623 = 'Moving'
  701 = 'Next'
  328 = 'Single Step'
  48 = 'Starting'
END_TEXTLIST

// ---- VISUs/Visualization.TcVIS
VISUALIZATION Visualization  // 2x2
END_VISUALIZATION

// ---- VISUs/Visu_XPlanarUtility.TcVIS
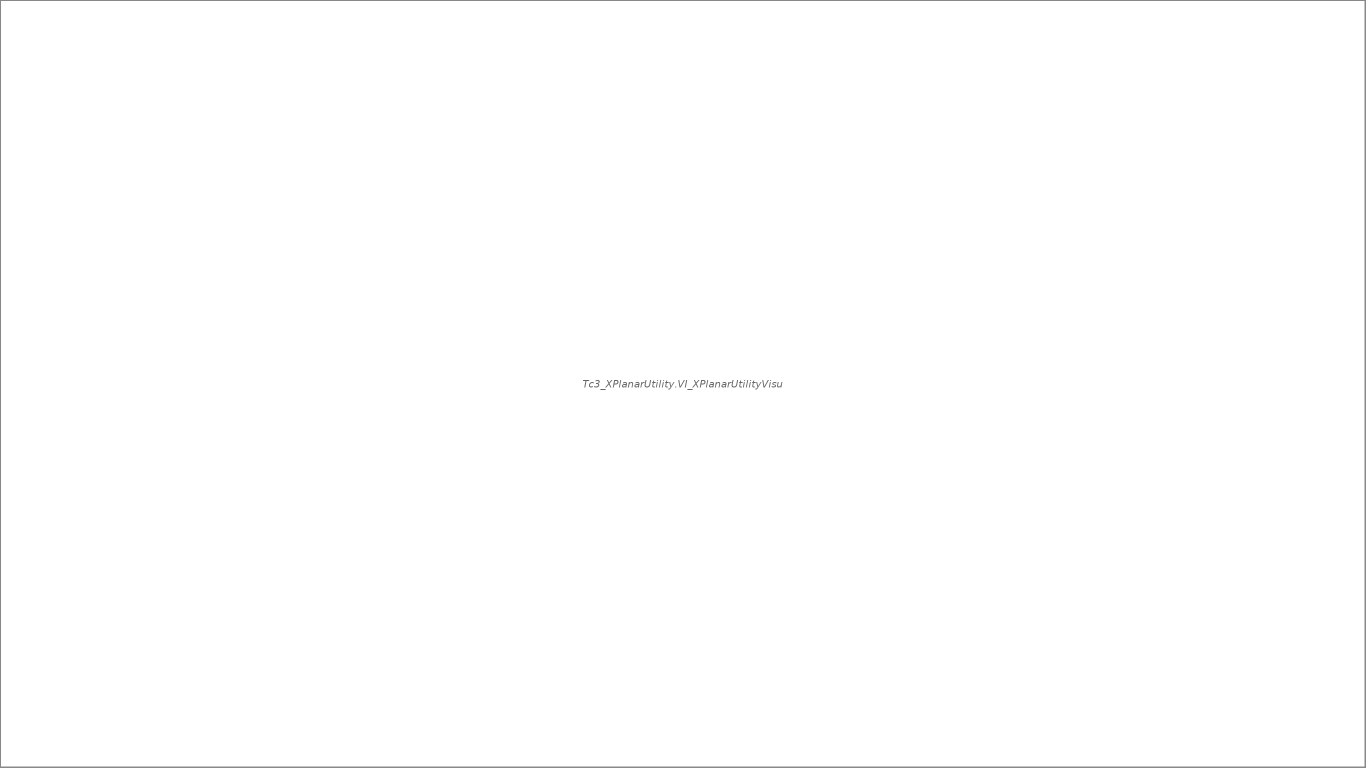
VISUALIZATION Visu_XPlanarUtility  // 1366x768
    Frame (0,0 1366x768)
        shows Tc3_XPlanarUtility.VI_XPlanarUtilityVisu()
END_VISUALIZATION
